FUNCTION_BLOCK ConveyorLSC EXTENDS ConveyorSC
VAR_OUTPUT
	lifterError AT %I* : BOOL;
	
	extended AT %I* : BOOL;
	retracted AT %I* : BOOL;
END_VAR
VAR	
	lifterEnable AT %Q* : BOOL := TRUE;
	lifterDirection AT %Q* : BOOL; //FALSE = up, TRUE = down
	lifterPulse AT %Q* : BOOL;
	lifterReset AT %Q* : BOOL;
END_VAR
VAR	
	lifterMode : (HOLD, LIFTER_EXTEND, LIFTER_RETRACT); 
	lifterPulser : TP; //pulses are assumed to be low-high-low
END_VAR

SUPER^();

lifterOverride();

lifterSequence();

METHOD backward : BOOL
VAR_INPUT
END_VAR
END_METHOD

METHOD extend : BOOL
VAR_INPUT
END_VAR
lifterMode := LIFTER_EXTEND;
END_METHOD

METHOD forward : BOOL
VAR_INPUT
END_VAR
END_METHOD

METHOD PROTECTED lifterOverride : BOOL
VAR_INPUT
END_VAR
IF
	(extended AND lifterMode = LIFTER_EXTEND) OR
	(retracted AND lifterMode = LIFTER_RETRACT)
THEN
	lifterMode := HOLD;
END_IF
END_METHOD

METHOD PROTECTED lifterSequence : BOOL
VAR_INPUT
END_VAR
VAR
	nextOp, prevOp : INT;
END_VAR
lifterPulser(IN:= , PT:= pulseWidth, Q=> , ET=> );
lifterPulser.IN := 
	lifterEnable AND 
	NOT lifterError AND 
	NOT lifterReset AND 
	( (lifterMode = LIFTER_EXTEND AND NOT extended) OR (lifterMode = LIFTER_RETRACT AND NOT retracted) ) AND
	lifterPulser.Q; //self-ending pulse

lifterPulse := lifterPulser.Q AND lifterPulser.ET < pulseWidth/2;
END_METHOD

METHOD reset : BOOL
VAR_INPUT
END_VAR
position := 0;
velocity := velocity; //no change

extend();
END_METHOD

METHOD retract : BOOL
VAR_INPUT
END_VAR
lifterMode := LIFTER_RETRACT;
END_METHOD

END_FUNCTION_BLOCK

(* stored: Version 1.1.0.1, ProductVersion 3.1.4024.11
   POU ConveyorLSC: Id {4e7826d2-4488-4b7a-b41d-13fd4487d89b}, SpecialFunc None
   Folder Private: Id {2314e23b-781d-4238-8176-f151798202cc}
   Folder Properties: Id {fff115d2-9fdf-4afc-9bdb-354b70770c2d}
   Folder Unused: Id {e0030328-56d3-4815-965e-93186e15fd6f}
   Method backward: Id {db97316a-330f-46e9-bc63-9ce67e31f10f}
   Method extend: Id {f68a79dc-ed79-43bf-a99b-a290f69cccbe}
   Method forward: Id {b9f1817e-75db-4f74-81eb-a7b6d0c52d27}
   Method lifterOverride: Id {1f87db49-62a1-4c44-98b6-f67e3ea2de36}
   Method lifterSequence: Id {dd26079e-18e0-4387-83ae-25d482a9933a}
   Method reset: Id {dcf20cf6-4c7e-4e08-a161-dbbbb376ac41}
   Method retract: Id {9aff9194-25b2-48ea-8527-e8dd9e3d287a} *)
